// TwinCAT 3 PLC project main
// ProgramVersion: 3.1.4024.0
// libraries:
//   Tc2_Standard, * (Beckhoff Automation GmbH)
//   Tc2_System, * (Beckhoff Automation GmbH)
//   Tc3_Module, * (Beckhoff Automation GmbH)
// project tree:
//   DUTs/ PID_Parameter_Strukt.TcDUT, PT1T2_Parameter_Strukt.TcDUT, System_Modus_Enum.TcDUT
//   GVLs/ IO.TcGVL
//   / PlcTask.TcTTO
//   POUs/ MAIN.TcPOU, PID_Regler.TcPOU, PT1T2_Prozess.TcPOU
// real-time tasks:
//   TASK PlcTask: cycle T#10ms, priority 20, ADS port 350
// I/O:
//   DEVICE Gerät 1 (EtherCAT), AmsNetId 10.180.42.21.2.1
//     Klemme 1 (EK1200) [EK1200-5000 EtherCAT Netzteil (2A E-Bus)]
//       Klemme 2 (EL1004) [EL1004 4K. Dig. Eingang 24V, 3ms]
//       Klemme 3 (EL2004) [EL2004 4K. Dig. Ausgang 24V, 0.5A]
//       Klemme 4 (EL3004) [EL3004 4K.Ana. Eingang  +/-10V]
//       Klemme 5 (EL4034) [EL4034 4K. Ana. Ausgang +/-10V, 12bit]
//       Klemme 6 (EK1110) [EK1110 EtherCAT-Verlängerung]
//     Klemme 7 (EK1100) [EK1100 EtherCAT-Koppler (2A E-Bus)]
//       Klemme 8 (EL3004) [EL3004 4K.Ana. Eingang  +/-10V]
//       Klemme 9 (EL5101) [EL5101 1K. Inc. Encoder 5V]
//       Klemme 10 (EL7342) [EL7342 2K. DC-Motor-Endstufe (50V, 3.5A)]
//       Klemme 11 (EL9011) [EL9011 Endklemme]
// variable links:
//   main/main Instance <-> Device 1 (EtherCAT)/Term 7 (EK1100)/Term 10 (EL7342)
//     PlcTask Outputs/IO.dc_MotorEnable <-> DCM Control Channel 2/Control/Enable
//     PlcTask Outputs/IO.dc_MotorVelocity <-> DCM Velocity Channel 2/Velocity
//   main/main Instance <-> Device 1 (EtherCAT)/Term 7 (EK1100)/Term 9 (EL5101)
//     PlcTask Inputs/IO.dc_Encoder <-> ENC Status compact/Counter value
//     PlcTask Inputs/IO.dc_OverflowBit <-> ENC Status compact/Status/Counter overflow
//     PlcTask Inputs/IO.dc_UnderflowBit <-> ENC Status compact/Status/Counter underflow

CONFIGURATION main
    RESOURCE PLC ON TwinCAT3
        TASK PlcTask(INTERVAL := T#10ms, PRIORITY := 20);
        PROGRAM MAIN WITH PlcTask : MAIN;
    END_RESOURCE
END_CONFIGURATION

// ---- DUTs/PID_Parameter_Strukt.TcDUT
TYPE PID_Parameter_Strukt :
STRUCT
	Kp :		REAL;
	Ti :		REAL;
	Td :		REAL;
	N :			REAL;
	ARW :		BOOL;
	Tr :		REAL;
	umin :		REAL;
	umax :		REAL;
END_STRUCT
END_TYPE

// ---- DUTs/PT1T2_Parameter_Strukt.TcDUT
TYPE PT1T2_Parameter_Strukt :
STRUCT
	K :			REAL;
	T1 :		REAL;
	T2 :		REAL;
END_STRUCT
END_TYPE

// ---- DUTs/System_Modus_Enum.TcDUT
{attribute 'qualified_only'}
{attribute 'strict'}
TYPE System_Modus_Enum :
(
	System_Init := 0,
	System_Run
);
END_TYPE

// ---- GVLs/IO.TcGVL
{attribute 'qualified_only'}
VAR_GLOBAL
	dc_Encoder			AT %I*	:UINT;
	dc_OverflowBit		AT %I* 	:BOOL;
	dc_UnderflowBit		AT %I*	:BOOL;
	
	dc_MotorEnable 		AT %Q* 	:BOOL;
	dc_MotorVelocity	AT %Q*	:INT;
END_VAR

// ---- POUs/MAIN.TcPOU
PROGRAM MAIN
VAR
	T :							REAL := 0.01;	
	K :							REAL := 10;
	PID_Parameter :				PID_Parameter_Strukt;
	Modus :						System_Modus_Enum := System_Modus_Enum.System_Init;
	PID_1 :						PID_Regler;
	
	r0 :						REAL := 0;	//Goal RPM
	dc_Encoder_old :			UINT := 0;
	dc_RPM : 					REAL := 0;	//DC Motor RPM (1 Rotation = 32,768 Impulses)
	u	:						REAL := 0;
	
	
	e0 :						REAL := 0;
END_VAR
//

CASE Modus OF
	System_Modus_Enum.System_Init:
	PID_Parameter.Kp := 100/K;
	PID_Parameter.Ti := 1;
	PID_Parameter.Td := 2;
	PID_Parameter.N := 10;
	PID_Parameter.umax := 10;
	PID_Parameter.umin := 0;
	PID_Parameter.ARW := TRUE;
	PID_Parameter.Tr := 0.1;
	Modus := System_Modus_Enum.System_Run
	;
	System_Modus_Enum.System_Run:
	IF ((IO.dc_Encoder - dc_Encoder_old) < 0) AND (Io.dc_OverflowBit = TRUE) THEN
		dc_RPM := ((65535 - dc_Encoder_old + IO.dc_Encoder) * (60*100/32768));
	ELSE
		dc_RPM := (INT_TO_REAL(IO.dc_Encoder - dc_Encoder_old) * (60.0*(1/T)/32768.0));
	END_IF;
	e0 := r0;
	PID_1(r1 := r0, y1 := 0, Modus := Modus, Param := PID_Parameter, T := T);
	dc_Encoder_old := IO.dc_Encoder;
	;

END_CASE

END_PROGRAM

// ---- POUs/PID_Regler.TcPOU
FUNCTION_BLOCK PID_Regler
VAR_INPUT
	r1 :			REAL;
	y1 :			REAL;
	Modus :		System_Modus_Enum;
	Param :		PID_Parameter_Strukt;
	T :			REAL;
END_VAR
VAR_OUTPUT
	u :			REAL;
END_VAR
VAR
	a0 :		REAL;
	b0 :		REAL;
	c0 :		REAL;

	rm :		REAL;
	ym :		REAL;
	u_temp :	REAL;
	up : 		REAL;
	ui :		REAL;
	ud :		REAL;
	uim :		REAL;
	udm :		REAL;
END_VAR

CASE Modus OF
	System_Modus_Enum.System_Init:
	c0 := (T*Param.Kp)/(2*Param.Ti);
	a0 := (Param.Td)/(Param.Td+Param.N*T);
	b0 := (Param.Kp*Param.Td*Param.N)/(Param.Td+Param.N*T);
	u := 0;
	rm := 0;
	ym := 0;
	up := 0;
	ui := 0;
	ud := 0;
	uim := 0;
	udm := 0;
	;
	System_Modus_Enum.System_Run:
	up := (r1-y1) * Param.Kp;
	IF Param.ARW = TRUE THEN
		ui := uim + c0*((r1-y1)+(rm-ym)) + (T/Param.Tr)*(u-u_temp);
	ELSE
		ui := uim + c0*((r1-y1)+(rm-ym));
	END_IF
	ud := b0 * ((r1-y1)-(rm-ym)) + a0 * udm;
	u := up + ui + ud;
	u_temp := u;
	IF u >= Param.umax THEN
		u := Param.umax;
	END_IF
	IF u <= Param.umin THEN
		u := Param.umin;
	END_IF
	rm := r1;
	ym := y1;
	uim := ui;
	udm := ud;
	;
END_CASE

END_FUNCTION_BLOCK

// ---- POUs/PT1T2_Prozess.TcPOU
FUNCTION_BLOCK PT1T2_Prozess
VAR_INPUT
	u :			REAL;
	Modus :		System_Modus_Enum;
	Param :		PT1T2_Parameter_Strukt;
	T :			REAL;
END_VAR
VAR_OUTPUT
	y :			REAL;
END_VAR
VAR
	alpha1 :	REAL;
	alpha2 :	REAL;
	a1 :		REAL;
	a2 :		REAL;
	b0 :		REAL;
	b1 :		REAL;
	b2 :		REAL;
	
	ym :		REAL;
	ymm :		REAL;
END_VAR

CASE Modus OF
	System_Modus_Enum.System_Init:
	alpha1 := T + Param.T1;
	alpha2 := T + Param.T2;
	a1 := 1;
	a2 := 2;
	b0 := (Param.K*T*T)/(alpha1*alpha2);
	a1 := -((Param.T1/alpha1)+(Param.T2/alpha2));
	a2 := (Param.T1*Param.T2)/(alpha1*alpha2);
	y := 0;
	ym := 0;
	ymm := 0;
	;
	System_Modus_Enum.System_Run:
	y := -a1 * ym - a2 *ymm + b0 * u;
	ymm := ym;
	ym := y;
	;
END_CASE

END_FUNCTION_BLOCK
